GLOBALCONSTANTS TCPool (* Global constants *)
  (* Standard: 61499-1; Description: Copyright (c) 2024 HR Agrartechnik GmbH This program and the accompanying materials are made available under the terms of the Eclipse Public License 2.0 which is available at https://www.eclipse.org/legal/epl-2.0/ SPDX-License-Identifier: EPL-2.0 *)
  (* Version 1.0, 2024-02-25, Franz Höpfinger, HR Agrartechnik GmbH *)
  PACKAGE Uebungen::const::TC;
  VAR_GLOBAL CONSTANT
    DE_NUM_DEVICE : UINT := 0;
  END_VAR
END_GLOBALCONSTANTS
